{attribute addProperty BoxType "AT2025-0250-0023"}
{attribute addProperty Id "A_0076_AT2001_5250_0017_AT2001_5250AT2001_C5E5984862678.25"}
{attribute addProperty CRC "1250746938"}
{attribute addProperty SizeInBites "626"}
{attribute addProperty SizeInBytes "78.25"}
TYPE A_0064_AT2025_0250_0023_AT2025_0250_4A8CE23A EXTENDS AT2025_BA5A9548 :
STRUCT
	{attribute addProperty Name "A_0076_AT2001_5250_0017_AT2001_5250"}
	A_0076_AT2001_5250_0017_AT2001_5250 : AT2001_C5E59848;
END_STRUCT
END_TYPE

(* stored: Version 1.2.0.0, ProductVersion 3.1.4024.9
   DUT A_0064_AT2025_0250_0023_AT2025_0250_4A8CE23A: Id {421c8dcc-c74f-497b-9915-7b47f7b97d3c} *)
